Staubli VAL3: stop.pgx

public program stop()
  local string l_sItem
begin
  //
  // QUIT KERNEL
  //
  // release
  cycleStatus:bMutex=false
  bQuit=true
  ? "STOPPING..."
  //
  if !bErrorLoading
    // reset all
    call plc:kill()
    call cycle_init()
    call remote_rstLight()
    l_sItem="kill"
    delay(1)
    call memory_onStop(l_sItem)
  endIf
  // BYE
  bQuit=false
  resetMotion()
  disablePower()
  $jogPage(true)
  title("")
  cls()
  //
end
